(*

## Short summary

An abstract class to implement methods which are not dependent on the data structure.

.. <legal notes>

legal notes
=================
| SPDX-FileCopyrightText: © 2024 ekvip automation GmbH <info@ekvip.de>
| SPDX-License-Identifier: Apache-2.0
| For details check: Apache-2.0_

.. _Apache-2.0: https://www.apache.org/licenses/LICENSE-2.0

.. </legal notes>



*)
FUNCTION_BLOCK ABSTRACT AbstractList EXTENDS AbstractCollection IMPLEMENTS CNM_CollectionInterfaces.IList, IListHelpers

(*

## Short summary

This method adds the given CNM_AbstractObject.IObject to the end of the list.
**Example:** 
Given a list that looks like this: (Head->) A B C (<- End),
calling append(D) on this list will place the D at the and,
making it the new End: (Head->) A B C D(<- End)

.. <legal notes>

legal notes
=================
| SPDX-FileCopyrightText: © 2022 ekvip automation GmbH <info@ekvip.de>
| SPDX-License-Identifier: Apache-2.0
| For details check: Apache-2.0_

.. _Apache-2.0: https://www.apache.org/licenses/LICENSE-2.0

.. </legal notes>



*)

METHOD ABSTRACT append :CNM_ReturnTypes.SingleExecutionResult
VAR_INPUT
	(*The object to be appended*)
	object		:CNM_AbstractObject.IObject;
END_VAR
END_METHOD

(*

## Short summary

This method adds all elements of the given collection to the end of this list.
**Example:**
For the list1: A B C and list2: D E F will be after ```list1.appendCollection(list2)```:
A B C D E F. Notice the elements are still in the same order they where befor on each subsection.

.. <legal notes>

legal notes
=================
| SPDX-FileCopyrightText: © 2022 ekvip automation GmbH <info@ekvip.de>
| SPDX-License-Identifier: Apache-2.0
| For details check: Apache-2.0_

.. _Apache-2.0: https://www.apache.org/licenses/LICENSE-2.0

.. </legal notes>


**Return:** ``CNM_ReturnTypes.SingleExecutionResult.SUCCESS``: new Container not needed / could be allocated and data was copied
	``CNM_ReturnTypes.SingleExecutionResult.ERROR``: new Container couldn't be allocated, container left unchanged
	``CNM_ReturnTypes.SingleExecutionResult.ABORTED``: NULL object or the list itself was passed

*)

METHOD ABSTRACT appendCollection :CNM_ReturnTypes.SingleExecutionResult
VAR_INPUT
	(*The collection to be appended*)
	collectionToAppend :CNM_CollectionInterfaces.ICollection;
END_VAR
END_METHOD

(*

## Short summary

This abstract property returns the class name of the concrete object, 
which is useful to check the class name for ``__DELETE``.

.. <legal notes>

legal notes
=================
| SPDX-FileCopyrightText: © 2022 ekvip automation GmbH <info@ekvip.de>
| SPDX-License-Identifier: Apache-2.0
| For details check: Apache-2.0_

.. _Apache-2.0: https://www.apache.org/licenses/LICENSE-2.0

.. </legal notes>

*)
PROPERTY ABSTRACT className : CNM_AbstractObject.ClassName
GET
END_GET
END_PROPERTY

(*

## Short summary

This property returns the last object in the first and removes it from the list. Can be seen as opposite of prepend.
**Example:**
On a list: (Head -->) A B C, list.dequeue will return A.
**Example 2:**
If you call prepend(x), a dequeue right after will return x.

.. <legal notes>

legal notes
=================
| SPDX-FileCopyrightText: © 2022 ekvip automation GmbH <info@ekvip.de>
| SPDX-License-Identifier: Apache-2.0
| For details check: Apache-2.0_

.. _Apache-2.0: https://www.apache.org/licenses/LICENSE-2.0

.. </legal notes>

*)

METHOD ABSTRACT dequeue :CNM_AbstractObject.IObject
END_METHOD

METHOD INTERNAL ABSTRACT instantSorting : CNM_ReturnTypes.SingleExecutionResult
VAR_INPUT
	order :SortingOrder;
	(*Optional: the comparator that should be used for the sort. Must not be changed while sort is in process*)
	comparator	: CNM_CollectionInterfaces.CNM_AbstractObject.IComparator := 0;
END_VAR
END_METHOD

(*

## Short summary

Inverts the order of the elements inside the object. Does not apply any kind of sorting, only reverses.

.. <legal notes>

legal notes
=================
| SPDX-FileCopyrightText: © 2022 ekvip automation GmbH <info@ekvip.de>
| SPDX-License-Identifier: Apache-2.0
| For details check: Apache-2.0_

.. _Apache-2.0: https://www.apache.org/licenses/LICENSE-2.0

.. </legal notes>



*)

METHOD ABSTRACT invert
END_METHOD

PROPERTY INTERNAL listChangeIndex : __XWORD
GET
listChangeIndex := THIS^.changesToCollection;
END_GET
SET
THIS^.changesToCollection := listChangeIndex;
END_SET
END_PROPERTY

(*

## Short summary

This property returns the last object in the list and removes it from the list. Can be seen as opposite of append.
**Example:**
On a list: (Head -->) A B C, list.pop will return C.
**Example 2:**
If you call append(x), a pop right after will return x.
May return a null pointer if list is empty

.. <legal notes>

legal notes
=================
| SPDX-FileCopyrightText: © 2022 ekvip automation GmbH <info@ekvip.de>
| SPDX-License-Identifier: Apache-2.0
| For details check: Apache-2.0_

.. _Apache-2.0: https://www.apache.org/licenses/LICENSE-2.0

.. </legal notes>

*)

METHOD ABSTRACT pop :CNM_AbstractObject.IObject
END_METHOD

(*

## Short summary

This method adds the given obejct to the end of the list.
**Example:** 
Given a list that looks like this: (Head->) A B C (<- End),
calling prepend(D) on this list will place the D at start,
making it the new Head: (Head->) D A B C (<- End)

.. <legal notes>

legal notes
=================
| SPDX-FileCopyrightText: © 2022 ekvip automation GmbH <info@ekvip.de>
| SPDX-License-Identifier: Apache-2.0
| For details check: Apache-2.0_

.. _Apache-2.0: https://www.apache.org/licenses/LICENSE-2.0

.. </legal notes>


**Return:** ``CNM_ReturnTypes.SingleExecutionResult.SUCCESS``: new Container not needed / could be allocated and data was copied
	``CNM_ReturnTypes.SingleExecutionResult.ERROR``: new Container couldn't be allocated, container left unchanged
	``CNM_ReturnTypes.SingleExecutionResult.ABORTED``: NULL object or the list itself was passed
	
*)

METHOD ABSTRACT prepend :CNM_ReturnTypes.SingleExecutionResult
VAR_INPUT
	(*The object to be prepended*)
	object	:CNM_AbstractObject.IObject;
END_VAR
END_METHOD

(*

## Short summary

This method adds all elements of the given collection to the start of this list. 
**Example:**
For the list1: A B C and list2: D E F will be after ```list1.prependCollection(list2)```:
D E F A B C. Notice the elements are still in the same order they where befor on each subsection.

.. <legal notes>

legal notes
=================
| SPDX-FileCopyrightText: © 2022 ekvip automation GmbH <info@ekvip.de>
| SPDX-License-Identifier: Apache-2.0
| For details check: Apache-2.0_

.. _Apache-2.0: https://www.apache.org/licenses/LICENSE-2.0

.. </legal notes>


**Return:** ``CNM_ReturnTypes.SingleExecutionResult.SUCCESS``: prepend was successful
	``CNM_ReturnTypes.SingleExecutionResult.ERROR``: collection to prepend didn't fit in old container, and new container couldn't be allocated
	``CNM_ReturnTypes.SingleExecutionResult.ABORTED``: NULL object or this arraylist was passed
	
*)

METHOD ABSTRACT prependCollection :CNM_ReturnTypes.SingleExecutionResult
VAR_INPUT
	(*The collection to be prepended*)
	collectionToPrepend :CNM_CollectionInterfaces.ICollection;
END_VAR
END_METHOD

(*

## Short summary

This method removes the first instance of the given object from the list.
Compares objects with hash value.
For example a Linked List: A B C A A D after remove(A) becomes: B C A A D

.. <legal notes>

legal notes
=================
| SPDX-FileCopyrightText: © 2022 ekvip automation GmbH <info@ekvip.de>
| SPDX-License-Identifier: Apache-2.0
| For details check: Apache-2.0_

.. _Apache-2.0: https://www.apache.org/licenses/LICENSE-2.0

.. </legal notes>



*)

METHOD ABSTRACT remove
VAR_INPUT
	(*The object to be removed from the list*)
	object		:CNM_AbstractObject.IObject;
END_VAR
END_METHOD

(*

## Short summary

This property returns strategies to sort the list in a desired order.

.. <legal notes>

legal notes
=================
| SPDX-FileCopyrightText: © 2024 ekvip automation GmbH <info@ekvip.de>
| SPDX-License-Identifier: Apache-2.0
| For details check: Apache-2.0_

.. _Apache-2.0: https://www.apache.org/licenses/LICENSE-2.0

.. </legal notes>

*)

PROPERTY sort : CNM_CollectionInterfaces.ISortable
GET
VAR_INST
	sortStrategy	:SortingStrategyExecutor(THIS^);
END_VAR
sort := sortStrategy;
END_GET
END_PROPERTY

METHOD INTERNAL ABSTRACT sorting : CNM_ReturnTypes.SingleExecutionState
VAR_INPUT
	execute :BOOL;
	order :SortingOrder;
	(*Optional: the comparator that should be used for the sort. Must not be changed while sort is in process*)
	comparator	: CNM_CollectionInterfaces.CNM_AbstractObject.IComparator := 0;
END_VAR
END_METHOD

END_FUNCTION_BLOCK

(* stored: Version 1.1.0.1, ProductVersion 3.1.4026.13
   POU AbstractList: Id {2b629813-b5c1-4f3a-82ef-fe84be1f4ca1}, SpecialFunc None
   Folder IInvertable: Id {7f740e60-66fa-4816-bf00-cbce0395643e}
   Folder IList: Id {62a4bb1e-aabc-410e-b597-79cdc9f3500f}
   Folder Protected: Id {644572fe-6d8d-43f7-a6d5-566aa702cc93}
   Method append: Id {2f94a678-a1e8-4421-b2a0-aef19bec4fec}
   Method appendCollection: Id {7683c611-f280-4c44-babd-251c57010f7c}
   Property className: Id {10582c55-db61-4083-9788-f04923a8f973}
   Get Get: Id {3aba1fdd-6e04-4c57-a747-a77d7163f8be}
   Method dequeue: Id {4cfb8acf-848a-4774-a99f-ffe05e6a908c}
   Method instantSorting: Id {95a9e5f9-fc11-490c-a487-db01b0bcc33e}
   Method invert: Id {0c44c772-9e28-4418-9948-67542427477b}
   Property listChangeIndex: Id {4a39c870-b4a9-4712-a4a5-4a389152f463}
   Get Get: Id {ab2d9eb5-0016-4ba9-ad68-3d99e1b0c30c}
   Set Set: Id {fe091184-098e-45b5-b549-0ab74d4dff83}
   Method pop: Id {e0bcabef-ab01-4f7f-a77c-39577aa93bae}
   Method prepend: Id {9b9a75f3-a9ed-488f-9162-4f48d410aef6}
   Method prependCollection: Id {cc72048c-bb34-4d7a-977e-a4c8e0d3f058}
   Method remove: Id {21c6097d-ebee-4bfc-801d-007662886f99}
   Property sort: Id {5f2cf59e-dae5-49ed-9433-37458a0b21e3}
   Get Get: Id {83598f82-e208-43a8-a1c1-1305ac702373}
   Method sorting: Id {51417ece-cc2a-4d25-a4e8-7a332bc48937} *)
